Fanuc KAREL source: kd00012.KL

-- PROVISIONAL review KL for V770-1; original PC SHA256 47a2d1fe3a1764c67d421aca8c419d3ab52dc74632f03eab623498edc0891194
-- Incomplete behavior may be omitted. Consult companion uncertainty JSON. Do not deploy.
PROGRAM KD00012
%NOLOCKGROUP
VAR
  I : INTEGER
  J : INTEGER
  B : BOOLEAN
  R : REAL
  S : STRING[80]
BEGIN
  -- UNRESOLVED_PC offsets 5-9; opcodes 9D,9D,1A
  -- UNRESOLVED_PC offsets 14-18; opcodes 7F
END KD00012
